(*
SPDX-FileCopyrightText: © 2026 Oleksandr Tiutyk <trofimich@gmail.com>
SPDX-License-Identifier: MIT
License: https://opensource.org/license/mit
*)

(*!
<summary>Receives compiler-initialized namespace metadata for Collections.</summary>
<description>
The exposed string remains library-owned and is read-only by contract. No allocation or runtime extraction occurs.
</description>
*)

FUNCTION_BLOCK INTERNAL NamespaceExtractor
VAR_OUTPUT
	(*!
<summary>Receives the library namespace from compiler initialization.</summary>
<description>
CurrentNamespace is populated by init_namespace and used as read-only diagnostic metadata. No runtime
extraction or allocation is performed.
</description>
*)

{attribute 'init_namespace'} 
	CurrentNamespace : STRING;	
END_VAR

END_FUNCTION_BLOCK

(* stored: Version 1.1.0.1
   POU NamespaceExtractor: Id {82c7e191-5376-479e-8d26-7381e8fb28dd}, SpecialFunc None *)
